FUNCTION_BLOCK MyWorker IMPLEMENTS I_Execute
VAR
	_exe: Execute(THIS^);
	_worker: LoopWorker;
	
END_VAR

PROPERTY Base : I_Worker
GET
Base := _worker.Base;
END_GET
END_PROPERTY

(*
If registered, this method will be executed cyclically.
*)
{attribute 'hide'}
METHOD Execute
VAR_INPUT
	nPhase	: INT;
END_VAR
_worker.Run();
END_METHOD

END_FUNCTION_BLOCK

(* stored: Version 1.1.0.1
   POU MyWorker: Id {f9b70b6f-0f98-480e-811a-e71080a78641}, SpecialFunc None
   Property Base: Id {e952360f-dfef-4fb8-a452-eb5e523b0fe0}
   Get Get: Id {b34ebdeb-e502-40f5-bc1b-850082b5dba9}
   Method Execute: Id {dcb0a034-e58a-4195-b0bf-d3704a369b16} *)
